SUBAPPLICATION mapping_Uebung_034a2 (* Numeric Value Input auf PWM Ausgang OctaOut_8_PWM *)
  (* Standard: 61499-2 *)
  (* Version 1.0, 2023-10-23, franz *)
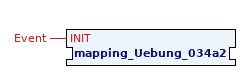
  EVENT_INPUT
    INIT;
  END_EVENT
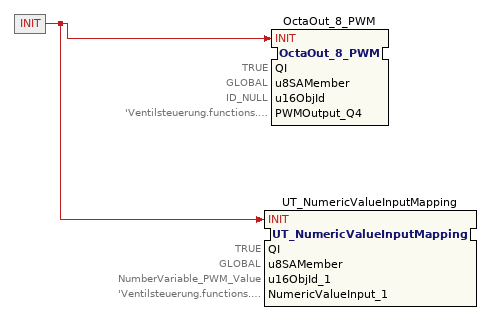
  FBS
    OctaOut_8_PWM : OctaOut_8_PWM(QI := TRUE, u8SAMember := GLOBAL, u16ObjId := ID_NULL, PWMOutput_Q4 := 'Ventilsteuerung.functions.PWMOutput_Q4');
    UT_NumericValueInputMapping : UT_NumericValueInputMapping(QI := TRUE, u8SAMember := GLOBAL, u16ObjId_1 := NumberVariable_PWM_Value, NumericValueInput_1 := 'Ventilsteuerung.functions.PWM_Value');
  END_FBS
  EVENT_CONNECTIONS
    INIT TO UT_NumericValueInputMapping.INIT;
    INIT TO OctaOut_8_PWM.INIT;
  END_CONNECTIONS
END_SUBAPPLICATION
